Staubli VAL3: Day6.dtx

string sInput
num nInput
lists lResult
  [0]
    string sString
num nResult
num nInput2
num nCounter[9]
